FUNCTION F_GetTransportTubeDevices : ST_TransportTubeDevices
VAR_INPUT
	eTransportTube : E_TransportTube;
END_VAR

CASE eTransportTube OF
E_TransportTube.BI1:
	F_GetTransportTubeDevices := GVL_TransportTubes.stBI1Dev;
E_TransportTube.BO4:
	F_GetTransportTubeDevices := GVL_TransportTubes.stBO4Dev;
END_CASE

END_FUNCTION

(* stored: Version 1.1.0.1, ProductVersion 3.1.4024.0
   POU F_GetTransportTubeDevices: Id {b2f27124-2dc4-4005-bbf3-37530c30c972}, SpecialFunc None *)
